{attribute addProperty BoxType "EL6201-0000-0017"}
{attribute addProperty Id "Slave_9A_DO0BIT10.12565Slave_9A_DO1BIT10.12566Slave_9A_DO2BIT10.12567Slave_9A_DO3BIT10.12568Slave_9B_DO0BIT10.12569Slave_9B_DO1BIT10.12570Slave_9B_DO2BIT10.12571Slave_9B_DO3BIT10.12572"}
{attribute addProperty CRC "281705881"}
{attribute addProperty SizeInBites "8"}
{attribute addProperty SizeInBytes "1"}
TYPE Slave_9_Outputs_10CA7D99 :
STRUCT
	{attribute addProperty Name "Slave_9A_DO0"}
	Slave_9A_DO0 : BIT;
	{attribute addProperty Name "Slave_9A_DO1"}
	Slave_9A_DO1 : BIT;
	{attribute addProperty Name "Slave_9A_DO2"}
	Slave_9A_DO2 : BIT;
	{attribute addProperty Name "Slave_9A_DO3"}
	Slave_9A_DO3 : BIT;
	{attribute addProperty Name "Slave_9B_DO0"}
	Slave_9B_DO0 : BIT;
	{attribute addProperty Name "Slave_9B_DO1"}
	Slave_9B_DO1 : BIT;
	{attribute addProperty Name "Slave_9B_DO2"}
	Slave_9B_DO2 : BIT;
	{attribute addProperty Name "Slave_9B_DO3"}
	Slave_9B_DO3 : BIT;
END_STRUCT
END_TYPE

(* stored: Version 1.2.0.0, ProductVersion 3.1.4024.9
   DUT Slave_9_Outputs_10CA7D99: Id {fe9ed5b7-20e3-4e57-af6b-c3d8d22776b4} *)
